// TIA Portal V21 export
TYPE "AxixAS_CFG_Type"
   STRUCT
      "xmm/degree" { S7_SetPoint := 'True'} : Bool;   // UM= Millimetri UNM= Gradi
      "xCurveS-L" { S7_SetPoint := 'True'} : Int;   // 0=curva TRAPEZIO 1=curva LOGARITMO 2=curva COS
      fJogSpeed { S7_SetPoint := 'True'} : Real := 10.0;   // Speed Jog movement (mm/sec) / Velocità JOG (mm/sec)
      fJogAcc { S7_SetPoint := 'True'} : Real := 10.0;   // Acc. jog movement (mm/sec^2) / Acc. JOG (mm/sec^2)
      fJogDec { S7_SetPoint := 'True'} : Real := 10.0;   // Dec. jog movement (mm/sec^2) / Dec. JOG (mm/sec^2)
      fVirt_EncWindPos { S7_SetPoint := 'True'} : Real := 1.0;   // Cycle end virtual encoder position window (mm) / Finestra di posizione encoder virtuale Stop (mm)
      fVirt_EncWindSpeed { S7_SetPoint := 'True'} : Real := 10.0;   // Cycle end virtual encoder speed window(mm/sec) / Finestra di velocità encoder virtuale Stop (mm/sec)
      fMotWindPos { S7_SetPoint := 'True'} : Real := 1.0;   // Cycle end motor position window (mm) / Finestra di posizione motore Stop (mm)
      fMotWindSpeed { S7_SetPoint := 'True'} : Real := 10.0;   // Cycle end motor speed window (mm/sec) / Finestra di velocità motore Stop (mm/sec)
      fMotWindPosBig { S7_SetPoint := 'True'} : Real := 30.0;   // Finestra Allargata di posizione motore Stop (mm)
      fMotAdvStopPosition { S7_SetPoint := 'True'} : Real := 30.0;   // Finestra per anticipo STOP al target virtuale
      fMaxErrEnc { S7_SetPoint := 'True'} : Real := 5.0;   // Max tracking value for alarm (mm) / Massimo valore inseguimento per allarme (mm)
      fKPpid_Pos { S7_SetPoint := 'True'} : Real := 1.0;   // PID Proportional constant / Anello Posizione Costante proporzionale PID
      fKPpidAcc_Pos { S7_SetPoint := 'True'} : Real := 1.0;   // Anello Posizione Costante proporzionale PID fase accelerazione
      fKPpidDec_Pos { S7_SetPoint := 'True'} : Real := 4.0;   // PID Proportional constant dec.phase / Anello Posizione Costante proporzionale PID fase decelerazione
      fKPpid_Vel { S7_SetPoint := 'True'} : Real := 1.0;   // Anello Velocità Costante proporzionale PID
      fKPpidAcc_Vel { S7_SetPoint := 'True'} : Real := 1.0;   // Anello Velocità Costante proporzionale PID fase accelerazione
      fKPpidDec_Vel { S7_SetPoint := 'True'} : Real := 1.0;   // Anello Velocità Costante proporzionale PID fase decelerazione
      fMinSpeed { S7_SetPoint := 'True'} : Real;   // Low limit speed requested (mm/sec) / Limite INF velocità richiesta (mm/sec)
      fMaxSpeed { S7_SetPoint := 'True'} : Real := 100.0;   // High speed limit (mm/sec) / Limite SUP velocità richiesta (mm/sec)
      fMaxAccRamp { S7_SetPoint := 'True'} : Real := 1200.0;   // Limite SUP Acc richiesta (mm/sec^2)
      fMaxDecRamp { S7_SetPoint := 'True'} : Real := 800.0;   // Limite SUP Dec richiesta (mm/sec^2)
      fFirstStepNepero { S7_SetPoint := 'True'} : Real := 6.0;   // Definisce gradino di ingresso Funzione Nepero
      "fAutoChangeS-Lvalue" { S7_SetPoint := 'True'} : Real;   // Cambio curva automatico se LOG -> TRA per spostamenti inferiori a...
      tBrakeDelay_Fwd { S7_SetPoint := 'True'} : Time := T#100ms;   // Valore timer sblocco freno avanti-salita
      tBrakeDelay_Bkw { S7_SetPoint := 'True'} : Time := T#100ms;   // Valore timer sblocco freno indietro-discesa
      tDriveOnReq { S7_SetPoint := 'True'} : Time := T#5s;   // Valore timer controllo mantenimento abilitazione inverter
      tCtrEndPos { S7_SetPoint := 'True'} : Time := T#1000ms;   // Valore timer allarme controllo fine posizionamento
   END_STRUCT;
END_TYPE
